FUNCTION_BLOCK TimeBreakdown
VAR_INPUT
	timesignal	:	ULINT;
END_VAR
VAR_OUTPUT	
	seconds	:	ULINT;
	milseconds	:	ULINT;
	micseconds	:	ULINT;
	nseconds	:	ULINT;
END_VAR
VAR	
END_VAR

nseconds := timesignal MOD 1000;

micseconds := (timesignal MOD 1000000)/1000;

milseconds := (timesignal MOD 1000000000)/1000000;

seconds := (timesignal MOD 1000000000000)/1000000000;

END_FUNCTION_BLOCK

(* stored: Version 1.1.0.1, ProductVersion 3.1.4024.12
   POU TimeBreakdown: Id {0cddfe48-76a7-4863-bc7a-1b9117520887}, SpecialFunc None *)
